(* PLC project FixtureLatch, Fixture plc-emu 0.1.0 *)
(* stored: creationDateTime 2025-11-20T00:00:00Z, modificationDateTime 2025-11-20T00:00:00Z, version 1.0, organization FixtureCo *)

PROGRAM Main_ST

END_PROGRAM

PROGRAM MainLadder

(* LD diagram, written out as Structured Text *)
END_PROGRAM

CONFIGURATION Config0
  VAR_GLOBAL
    StartPB AT %IX0.0 : BOOL;
    StopPB AT %IX0.1 : BOOL;
    MotorCmd : BOOL;
    MotorOut AT %QX0.0 : BOOL;
    StatusLamp AT %QX0.1 : BOOL;
  END_VAR
  RESOURCE Resource1 ON PLC
    TASK CyclicTask(INTERVAL := T#100ms, PRIORITY := 1);
  END_RESOURCE
END_CONFIGURATION
